FUNCTION_BLOCK AerateOC (* CAT Function Block Type *)
  (* Standard: 61499-2 *)
  (* Version 0.0, 6/7/2026, Schneider Electric, template *)
  PACKAGE SE.Nereda;
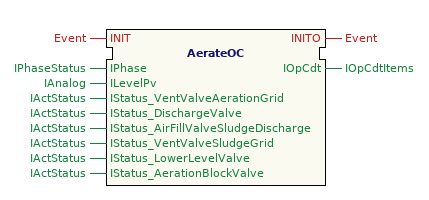
  EVENT_INPUT
    INIT;
  END_EVENT
  EVENT_OUTPUT
    INITO;
  END_EVENT
  SOCKETS
    IPhase : IPhaseStatus;
    ILevelPv : IAnalog;
    IStatus_VentValveAerationGrid : IActStatus;
    IStatus_DischargeValve : IActStatus;
    IStatus_AirFillValveSludgeDischarge : IActStatus;
    IStatus_VentValveSludgeGrid : IActStatus;
    IStatus_LowerLevelValve : IActStatus;
    IStatus_AerationBlockValve : IActStatus;
  END_SOCKETS
  PLUGS
    IOpCdt : IOpCdtItems;
  END_PLUGS
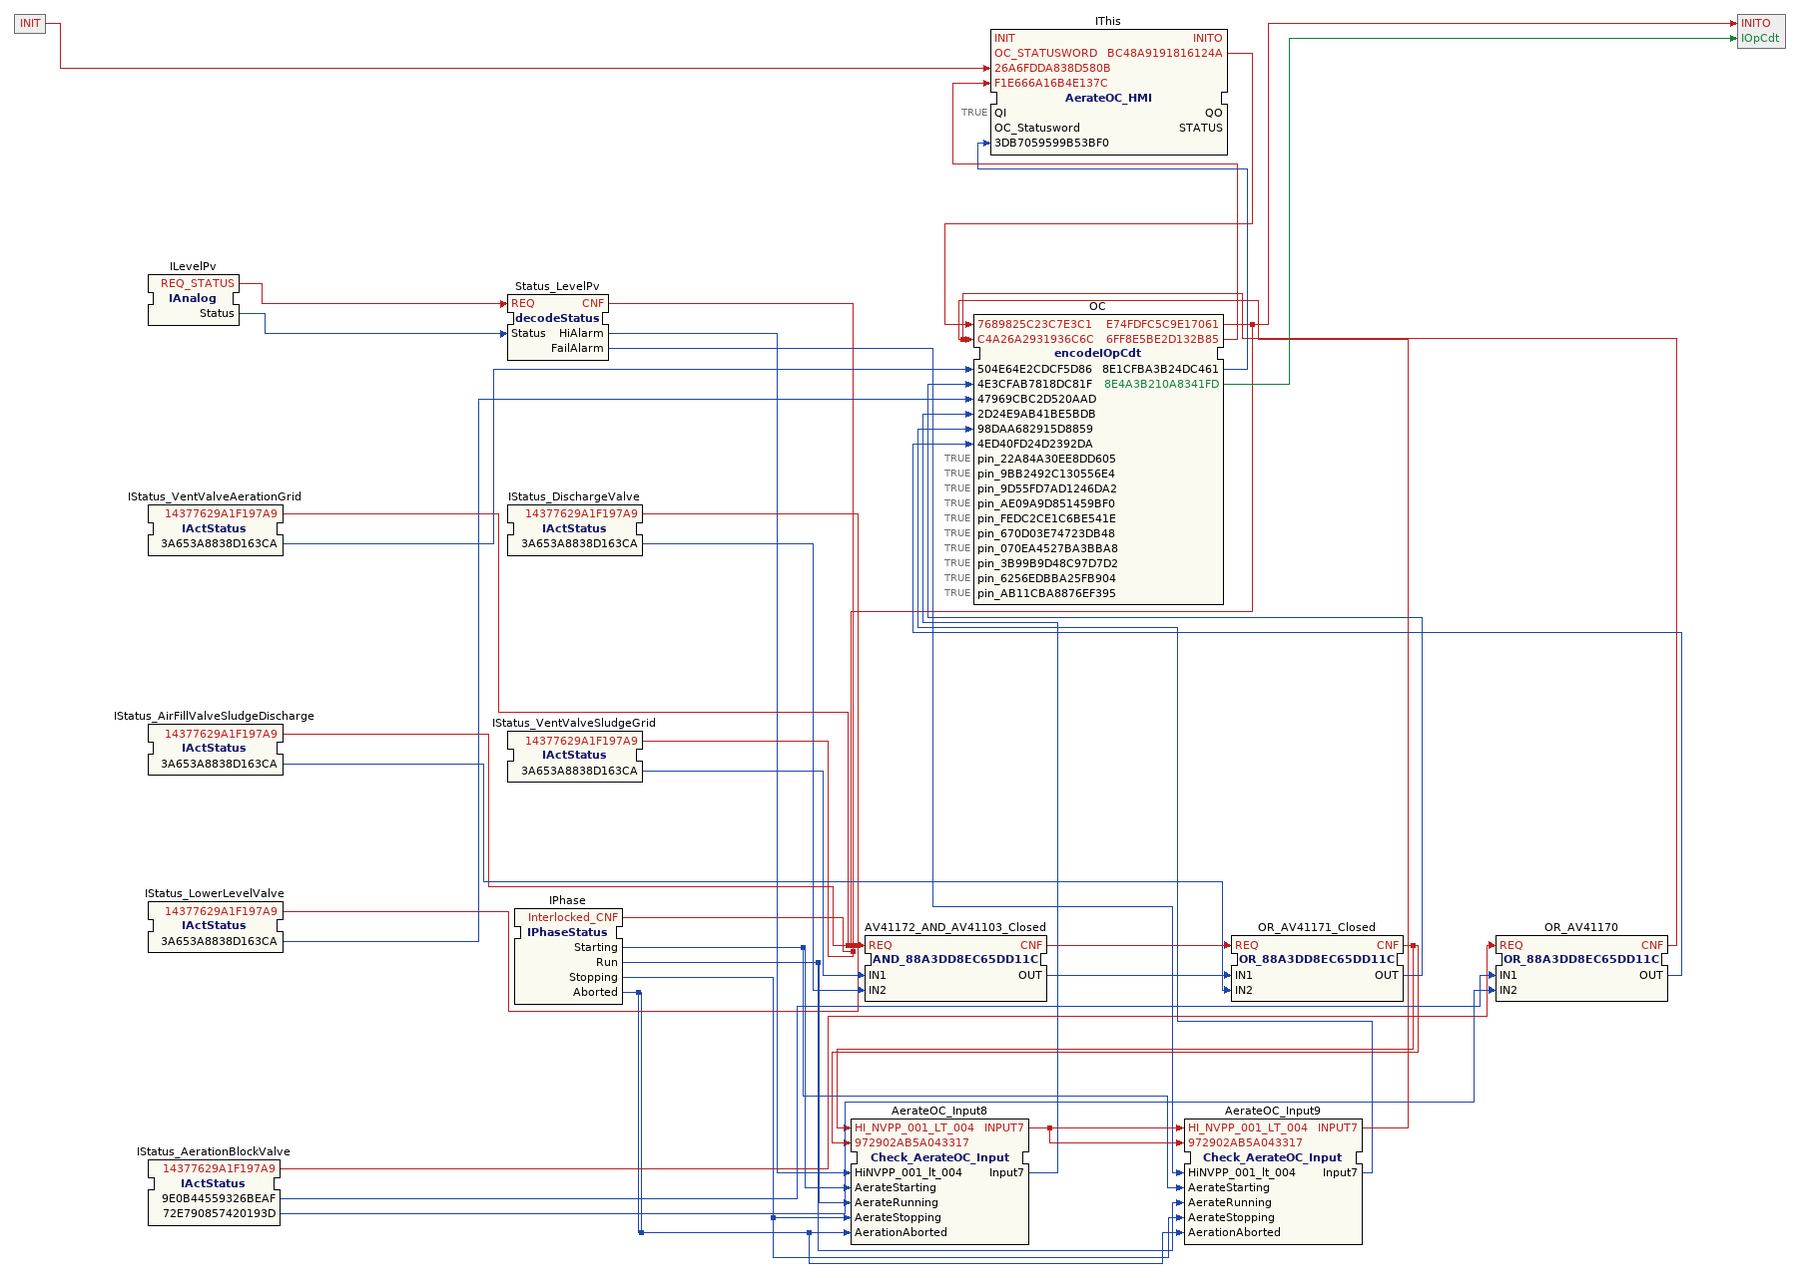
  (* 01 - FUNCTIONNAL INPUT INTERFACE *)
  (* 00 - INITIALIZATION *)
  (* 05 - LOGIC *)
  (* 06 - HMI INTERFACE *)
  (* 03 - FIELD INTERFACE *)
  (* Operating Condition Status *)
  (* Created by : Nouriddin OUECHEN 2026 *)
  (* 02 - FUNCTIONNAL OUTPUT INTERFACE *)
  (* Operating conditions : 2. Aeration Block Valve AV-41-170 is available or open 3. Vent valve aeration grid AV41107 is closed 6. Air fill valve sludge discharge AV41171 is closed OR (air vent valve AV41172 AND sludge discharge valve AV41103 are closed) 7. Lower level valve AV41102 is closed. 8. NOT (High level (aeration) in reactor 41LT1005) OR phase ‘aerate’ (‘starting’ or ‘RUN’ or ‘stopping’)) 9. Level measurement 41LT1005 available OR phase ‘aerate’ (‘starting’ or ‘RUN’ or ‘stopping’)) *)
  (* Actuators Tags : - Feed valve :                                  AV4x101 - Lower level valve :                        AV4x102 - Air fill valve sludge discharge :    AV4x171 - Chemicals valve :                         AV4x108 - Discharge valve :                         AV4x103 - Vent aeration grid valve :             AV4x107 - Vent sludge grid valve :               AV4x172 *)
  FBS
    OC : encodeIOpCdt(pin_22A84A30EE8DD605 := TRUE, pin_9BB2492C130556E4 := TRUE, pin_9D55FD7AD1246DA2 := TRUE, pin_AE09A9D851459BF0 := TRUE, pin_FEDC2CE1C6BE541E := TRUE, pin_670D03E74723DB48 := TRUE, pin_070EA4527BA3BBA8 := TRUE, pin_3B99B9D48C97D7D2 := TRUE, pin_6256EDBBA25FB904 := TRUE, pin_AB11CBA8876EF395 := TRUE); (* You set the operating conditions. For the inputs that are not used set a constant to TRUE. *)
    IThis : AerateOC_HMI(QI := TRUE);
    Status_LevelPv : decodeStatus; {SET_ATTRIBUTE(Configuration.Component.HideUnusedPorts, )}
    AerateOC_Input8 : Check_AerateOC_Input;
    AerateOC_Input9 : Check_AerateOC_Input;
    AV41172_AND_AV41103_Closed : AND_88A3DD8EC65DD11C; {SET_ATTRIBUTE(Configuration.GenericFBType.InterfaceParams, Runtime.Standard#CNT:=2;OUT:BOOL)}
    OR_AV41171_Closed : OR_88A3DD8EC65DD11C; {SET_ATTRIBUTE(Configuration.GenericFBType.InterfaceParams, Runtime.Standard#CNT:=2;OUT:BOOL)}
    OR_AV41170 : OR_88A3DD8EC65DD11C; {SET_ATTRIBUTE(Configuration.GenericFBType.InterfaceParams, Runtime.Standard#CNT:=2;OUT:BOOL)}
  END_FBS
  EVENT_CONNECTIONS
    INIT TO IThis.26A6FDDA838D580B;
    ILevelPv.REQ_STATUS TO Status_LevelPv.REQ;
    Status_LevelPv.CNF TO AV41172_AND_AV41103_Closed.REQ;
    IStatus_VentValveAerationGrid.14377629A1F197A9 TO AV41172_AND_AV41103_Closed.REQ;
    IStatus_DischargeValve.14377629A1F197A9 TO AV41172_AND_AV41103_Closed.REQ;
    IPhase.Interlocked_CNF TO AV41172_AND_AV41103_Closed.REQ;
    AerateOC_Input8.INPUT7 TO AerateOC_Input9.HI_NVPP_001_LT_004;
    AerateOC_Input8.INPUT7 TO AerateOC_Input9.972902AB5A043317;
    IThis.BC48A9191816124A TO OC.7689825C23C7E3C1;
    OC.E74FDFC5C9E17061 TO INITO;
    OC.E74FDFC5C9E17061 TO AV41172_AND_AV41103_Closed.REQ;
    OC.6FF8E5BE2D132B85 TO IThis.F1E666A16B4E137C;
    AerateOC_Input9.INPUT7 TO OC.C4A26A2931936C6C;
    AV41172_AND_AV41103_Closed.CNF TO OR_AV41171_Closed.REQ;
    IStatus_AirFillValveSludgeDischarge.14377629A1F197A9 TO AV41172_AND_AV41103_Closed.REQ;
    IStatus_VentValveSludgeGrid.14377629A1F197A9 TO AV41172_AND_AV41103_Closed.REQ;
    IStatus_LowerLevelValve.14377629A1F197A9 TO AV41172_AND_AV41103_Closed.REQ;
    OR_AV41171_Closed.CNF TO AerateOC_Input8.HI_NVPP_001_LT_004;
    OR_AV41171_Closed.CNF TO AerateOC_Input8.972902AB5A043317;
    IStatus_AerationBlockValve.14377629A1F197A9 TO OR_AV41170.REQ;
    OR_AV41170.CNF TO OC.C4A26A2931936C6C;
  END_CONNECTIONS
  DATA_CONNECTIONS
    ILevelPv.Status TO Status_LevelPv.Status;
    Status_LevelPv.HiAlarm TO AerateOC_Input8.HiNVPP_001_lt_004;
    Status_LevelPv.FailAlarm TO AerateOC_Input9.HiNVPP_001_lt_004;
    IPhase.Starting TO AerateOC_Input8.AerateStarting;
    IPhase.Starting TO AerateOC_Input9.AerateStarting;
    IPhase.Run TO AerateOC_Input8.AerateRunning;
    IPhase.Run TO AerateOC_Input9.AerateRunning;
    IPhase.Stopping TO AerateOC_Input8.AerateStopping;
    IPhase.Stopping TO AerateOC_Input9.AerateStopping;
    IPhase.Aborted TO AerateOC_Input8.AerationAborted;
    IPhase.Aborted TO AerateOC_Input9.AerationAborted;
    OC.8E1CFBA3B24DC461 TO IThis.3DB7059599B53BF0;
    IStatus_VentValveAerationGrid.3A653A8838D163CA TO OC.504E64E2CDCF5D86;
    AV41172_AND_AV41103_Closed.OUT TO OR_AV41171_Closed.IN1;
    OR_AV41171_Closed.OUT TO OC.4E3CFAB7818DC81F;
    IStatus_AirFillValveSludgeDischarge.3A653A8838D163CA TO OR_AV41171_Closed.IN2;
    IStatus_VentValveSludgeGrid.3A653A8838D163CA TO AV41172_AND_AV41103_Closed.IN1;
    IStatus_DischargeValve.3A653A8838D163CA TO AV41172_AND_AV41103_Closed.IN2;
    IStatus_LowerLevelValve.3A653A8838D163CA TO OC.47969CBC2D520AAD;
    AerateOC_Input8.Input7 TO OC.2D24E9AB41BE5BDB;
    AerateOC_Input9.Input7 TO OC.98DAA682915D8859;
    IStatus_AerationBlockValve.9E0B44559326BEAF TO OR_AV41170.IN1;
    IStatus_AerationBlockValve.72E790857420193D TO OR_AV41170.IN2;
    OR_AV41170.OUT TO OC.4ED40FD24D2392DA;
  END_CONNECTIONS
  ADAPTER_CONNECTIONS
    OC.8E4A3B210A8341FD TO IOpCdt;
  END_CONNECTIONS
END_FUNCTION_BLOCK
